Staubli VAL3: decodeMsgHeader.pgx

public program decodeMsgHeader(num& x_nMsgRecvState (dimensions=1))
  local num l_nRetVal
begin
  // Copyright (c) 2016, Ocado Technology - Robotics Research Team
  //
  // Licensed under the Apache License, Version 2.0 (the "License");
  // you may not use this file except in compliance with the License.
  // You may obtain a copy of the License at
  //
  //     http://www.apache.org/licenses/LICENSE-2.0
  //
  // Unless required by applicable law or agreed to in writing, software
  // distributed under the License is distributed on an "AS IS" BASIS,
  // WITHOUT WARRANTIES OR CONDITIONS OF ANY KIND, either express or implied.
  // See the License for the specific language governing permissions and
  // limitations under the License.



  // decode message into generic message first
  l_nRetVal=fromBinary(rosGenericMsg.prefix.nData,4,"-4l",rosGenericMsg.prefix.nLength)
  if (l_nRetVal!=1)
    // error decoding prefix, reset state machine
    x_nMsgRecvState=0
    return
  endIf
  l_nRetVal=fromBinary(rosGenericMsg.header.nData,4,"-4l",rosGenericMsg.header.nMsgType)
  if (l_nRetVal!=1)
    // error decoding header (msg type), reset state machine
    x_nMsgRecvState=0
    return
  endIf
  l_nRetVal=fromBinary(rosGenericMsg.header.nData[4],4,"-4l",rosGenericMsg.header.nCommType)
  if (l_nRetVal!=1)
    // error decoding header (comm type), reset state machine
    x_nMsgRecvState=0
    return
  endIf
  l_nRetVal=fromBinary(rosGenericMsg.header.nData[8],4,"-4l",rosGenericMsg.header.nReplyCode)
  if (l_nRetVal!=1)
    // error decoding header (reply code), reset state machine
    x_nMsgRecvState=0
    return
  endIf

  // no errors detected whilst decoding prefix and header
  // move on to state 2: receive msg body
  x_nMsgRecvState=2
end
